FUNCTION_BLOCK PUBLIC TcoRtc IMPLEMENTS ITcoRtc
VAR
	{attribute 'hide'}
	_LocalTime 							:	Tc2_Utilities.TIMESTRUCT;
	{attribute 'hide'}
	_UTCTime 							:	Tc2_Utilities.TIMESTRUCT;
	{attribute 'hide'}
	_LocalTimeDT						:	DATE_AND_TIME;
	{attribute 'hide'}
	_UTCTimeDT 							:	DATE_AND_TIME;
	{attribute 'hide'}
	_timeTick							: 	Tc2_EtherCAT.T_DCTIME64;
	
	
	{attribute 'hide'}
	_state								:	UINT;

	{attribute 'hide'}
	_NT_GetLocalTime					: 	Tc2_Utilities.NT_GetTime;
	{attribute 'hide'}
	_FB_TzSpecificLocalTimeToSystemTime :	Tc2_Utilities.FB_TzSpecificLocalTimeToSystemTime;
	{attribute 'hide'}
	_offset								:	ULINT;
_isValid : BOOL := TRUE;

_RtcSynchParams : RtcSynchParams;
END_VAR

PROPERTY IsValid : BOOL
GET
IsValid := _isValid;
END_GET
END_PROPERTY

METHOD NowLocal : DATE_AND_TIME
IF _isValid THEN
	NowLocal := _LocalTimeDT;
END_IF
END_METHOD

METHOD NowLocalAsTIMESTRUCT : Tc2_Utilities.TIMESTRUCT
IF _isValid THEN
	NowLocalAsTIMESTRUCT := _LocalTime;
END_IF
END_METHOD

METHOD NowUTC : DATE_AND_TIME
IF _isValid THEN
	NowUTC := _UTCTimeDT;
END_IF
END_METHOD

METHOD NowUTCAsTIMESTRUCT : Tc2_Utilities.TIMESTRUCT
IF _isValid THEN
	NowUTCAsTIMESTRUCT := _UTCTime;
END_IF
END_METHOD

PROPERTY RtcSynchParams : RtcSynchParams
GET
RtcSynchParams :=  _RtcSynchParams;
END_GET
SET
IF RtcSynchParams.synchContextIdentity <> 0 AND _RtcSynchParams.synchContextIdentity = 0 THEN
	_RtcSynchParams.synchContextIdentity := RtcSynchParams.synchContextIdentity; 
	_state := 0;
END_IF

IF _RtcSynchParams.synchContextIdentity <> 0 AND _RtcSynchParams.synchContextIdentity = RtcSynchParams.synchContextIdentity THEN
	_RtcSynchParams.doSynch := RtcSynchParams.doSynch;
	_RtcSynchParams.syncAmsId := RtcSynchParams.syncAmsId;
	_RtcSynchParams.syncPeriod := RtcSynchParams.syncPeriod;
END_IF
END_SET
END_PROPERTY

METHOD TickClock : ULINT
TickClock := Tc2_EtherCAT.F_GetActualDcTime64();
END_METHOD

METHOD Update
//VAR_INPUT
//	inContextIdentity	: ULINT;
//END_VAR
VAR	
	_TimeZoneID							:	Tc2_Utilities.E_TimeZoneID;
END_VAR
//IF _state = 0 THEN
//	_NT_GetLocalTime(NETID := '127.0.0.1.1.1', START := TRUE);
//	IF _NT_GetLocalTime.BUSY AND NOT _NT_GetLocalTime.ERR THEN 
//		_state := _state + 10;
//	END_IF
//END_IF
	
//IF _state = 10 THEN
//	_NT_GetLocalTime(START := FALSE);
//	IF NOT _NT_GetLocalTime.BUSY AND NOT _NT_GetLocalTime.ERR THEN 
//		_state := _state + 10;
//	END_IF
//END_IF

//IF _state = 20 THEN
	_NT_GetLocalTime(START := FALSE);
	_NT_GetLocalTime(NETID := '127.0.0.1.1.1', START := TRUE);
	_NT_GetLocalTime(START := FALSE);
		
	_LocalTime := _NT_GetLocalTime.TIMESTR;
	_LocalTimeDT := Tc2_Utilities.SYSTEMTIME_TO_DT(_NT_GetLocalTime.TIMESTR);

	IF RTC._isValid THEN
		_FB_TzSpecificLocalTimeToSystemTime(in 		:=	_LocalTime,
											tzInfo 	:=	RTC._TimeZoneInformation,
											out		=>	_UTCTime,
											eTzID	=>	_TimeZoneID);

		_UTCTimeDT := Tc2_Utilities.SYSTEMTIME_TO_DT(_UTCTime);
	END_IF
	_state := 0;
	
//	_timeTick :=  Tc2_EtherCAT.F_GetActualDcTime64(); 


//END_IF
END_METHOD

END_FUNCTION_BLOCK

(* stored: Version 1.1.0.1, ProductVersion 3.1.4024.6
   POU TcoRtc: Id {44984f17-252b-05a5-3965-3576c168912a}, SpecialFunc None
   Property IsValid: Id {0b73d0fb-6a2d-0c9e-3da7-384d62e156b5}
   Get Get: Id {f1495f6e-f4ab-08bd-138d-164d6df2166a}
   Method NowLocal: Id {ba634665-0212-047c-1c1d-6ebb5a5f30b5}
   Method NowLocalAsTIMESTRUCT: Id {e9fe0ffa-a159-017e-3bd5-9e67f37e7fa9}
   Method NowUTC: Id {34a4b82c-d3a2-0332-3148-6e27e32eec88}
   Method NowUTCAsTIMESTRUCT: Id {6c922f94-0952-07e6-0cac-83326b01c28c}
   Property RtcSynchParams: Id {b04a98c0-f35d-0885-0560-168bc0d55c2c}
   Get Get: Id {b4cdc5ff-8d88-0b4c-0de5-bfaa3fd2182c}
   Set Set: Id {757baeb2-5395-046e-24d5-a8962693357c}
   Method TickClock: Id {1cdfb043-4f81-0904-37ac-2a0334c75a58}
   Method Update: Id {0bf459e2-db45-0e5b-3d87-31081b5a02e2} *)
